TYPE s_DataSampleGatelength :
STRUCT
	gateLength	: LREAL;
	setDate		: STRING;
END_STRUCT
END_TYPE

(* stored: Version 1.1.0.1, ProductVersion 3.1.4024.11
   DUT s_DataSampleGatelength: Id {92a54464-5105-4c2b-b771-3da6a05e250a} *)
